PROGRAM MAIN
VAR
END_VAR

END_PROGRAM

(* stored: Version 1.1.0.1
   POU MAIN: Id {f4440f22-a180-4d20-882d-38619bc58b30} *)
